(* IEC 61131-3 sources: ST_L/Practice/04_FunctionBlock, 3 files *)

(* ---- 04_01_CounterFB.st ---- *)
(* ============================================================================
 * 文件: 04_01_CounterFB.st
 * 章节: 第7章 - 功能块
 * 描述: 计数器功能块
 * 学习目标: 掌握功能块的定义和实例化
 * ============================================================================ *)

(* ============================================================================
 * 功能块: Counter
 * 功能: 双向计数器，支持递增/递减计数
 * ============================================================================ *)
FUNCTION_BLOCK Counter
VAR_INPUT
    enable : BOOL := TRUE;           // 使能
    preset : INT := 100;             // 预设值
    increment : BOOL;                // 递增触发
    decrement : BOOL;                // 递减触发
    reset : BOOL;                    // 复位
END_VAR

VAR_OUTPUT
    currentValue : INT;              // 当前计数值
    done : BOOL;                     // 计数完成标志
    underflow : BOOL;                // 欠流标志
    overflow : BOOL;                 // 溢出标志
END_VAR

VAR
    lastInc : BOOL := FALSE;         // 上次递增状态
    lastDec : BOOL := FALSE;         // 上次递减状态
    lastReset : BOOL := FALSE;       // 上次复位状态
END_VAR

BEGIN
    (* 检测递增上升沿 *)
    IF increment AND NOT lastInc THEN
        IF enable THEN
            IF currentValue < 32767 THEN
                currentValue := currentValue + 1;
            ELSE
                overflow := TRUE;
            END_IF
        END_IF
    END_IF;

    (* 检测递减上升沿 *)
    IF decrement AND NOT lastDec THEN
        IF enable THEN
            IF currentValue > -32768 THEN
                currentValue := currentValue - 1;
            ELSE
                underflow := TRUE;
            END_IF
        END_IF
    END_IF;

    (* 检测复位上升沿 *)
    IF reset AND NOT lastReset THEN
        currentValue := 0;
        done := FALSE;
        overflow := FALSE;
        underflow := FALSE;
    END_IF;

    (* 更新完成状态 *)
    done := (currentValue >= preset);

    (* 保存上次状态 *)
    lastInc := increment;
    lastDec := decrement;
    lastReset := reset;
END_FUNCTION_BLOCK

(* ============================================================================
 * 功能块: UpCounter (递增计数器简化版)
 * ============================================================================ *)
FUNCTION_BLOCK UpCounter
VAR_INPUT
    enable : BOOL := TRUE;
    preset : INT := 100;
    count : BOOL;                    // 计数脉冲
    reset : BOOL;
END_VAR

VAR_OUTPUT
    q : BOOL;                        // 达到预设值
    cv : INT;                        // 当前值
END_VAR

VAR
    lastCount : BOOL := FALSE;
END_VAR

BEGIN
    (* 边沿检测 *)
    IF count AND NOT lastCount THEN
        IF enable AND NOT q THEN
            cv := cv + 1;
        END_IF
    END_IF;

    (* 复位 *)
    IF reset THEN
        cv := 0;
    END_IF;

    (* 输出 *)
    q := (cv >= preset);
    lastCount := count;
END_FUNCTION_BLOCK

(* ============================================================================
 * 功能块: DownCounter (递减计数器简化版)
 * ============================================================================ *)
FUNCTION_BLOCK DownCounter
VAR_INPUT
    enable : BOOL := TRUE;
    preset : INT := 10;
    count : BOOL;                    // 计数脉冲
    reset : BOOL;
END_VAR

VAR_OUTPUT
    q : BOOL;                        // 计数值减到0
    cv : INT;                        // 当前值
END_VAR

VAR
    lastCount : BOOL := FALSE;
END_VAR

BEGIN
    (* 边沿检测 *)
    IF count AND NOT lastCount THEN
        IF enable AND NOT q THEN
            IF cv > 0 THEN
                cv := cv - 1;
            END_IF
        END_IF
    END_IF;

    (* 复位 *)
    IF reset THEN
        cv := preset;
    END_IF;

    (* 输出 *)
    q := (cv <= 0);
    lastCount := count;
END_FUNCTION_BLOCK

(* ============================================================================
 * 功能块: CounterWithRate (带速率的计数器)
 * ============================================================================ *)
FUNCTION_BLOCK CounterWithRate
VAR_INPUT
    enable : BOOL := TRUE;
    preset : INT := 1000;
    pulse : BOOL;                    // 计数脉冲
    reset : BOOL;
    presetValue : INT;              // 可变预设值
END_VAR

VAR_OUTPUT
    current : INT;                   // 当前值
    done : BOOL;
    rate : REAL;                    // 计数速率 (次/秒)
END_VAR

VAR
    lastPulse : BOOL := FALSE;
    pulseCount : INT := 0;
    lastSecond : TIME := T#0s;
    currentSecond : TIME;
    rateTimer : TON;
END_VAR

BEGIN
    (* 检测脉冲 *)
    IF pulse AND NOT lastPulse THEN
        IF enable THEN
            current := current + 1;
            pulseCount := pulseCount + 1;
        END_IF
    END_IF;

    lastPulse := pulse;

    (* 复位 *)
    IF reset THEN
        current := 0;
        pulseCount := 0;
    END_IF;

    (* 计算速率 *)
    rateTimer(IN := enable, PT := T#1s);
    IF rateTimer.Q THEN
        rate := INT_TO_REAL(pulseCount);
        pulseCount := 0;
        rateTimer(IN := FALSE);
        rateTimer(IN := TRUE, PT := T#1s);
    END_IF;

    (* 完成标志 *)
    IF presetValue > 0 THEN
        done := (current >= presetValue);
    ELSE
        done := (current >= preset);
    END_IF
END_FUNCTION_BLOCK

(* ============================================================================
 * 程序: CounterDemo
 * 功能: 计数器功能块演示
 * ============================================================================ *)
PROGRAM CounterDemo
VAR
    (* 计数器实例 *)
    mainCounter : Counter;
    partCounter : UpCounter;
    batchCounter : DownCounter;
    rateCounter : CounterWithRate;

    (* 输入信号模拟 *)
    bPulse : BOOL := FALSE;
    bButton : BOOL := FALSE;

    (* 输出显示 *)
    iCount : INT;
    bDone : BOOL;
    rRate : REAL;

    (* 测试循环 *)
    i : INT;
END_VAR

BEGIN
    // ==========================================================================
    // 1. 基本计数器演示
    // ==========================================================================

    mainCounter(
        enable := TRUE,
        preset := 10,
        increment := bButton,
        decrement := FALSE,
        reset := FALSE
    );

    // 模拟10次计数
    FOR i := 1 TO 10 DO
        bButton := TRUE;
        mainCounter(
            enable := TRUE,
            preset := 10,
            increment := bButton,
            decrement := FALSE,
            reset := FALSE
        );
        bButton := FALSE;
    END_FOR;

    iCount := mainCounter.currentValue;  // 10
    bDone := mainCounter.done;           // TRUE

    // ==========================================================================
    // 2. 递增计数器演示
    // ==========================================================================

    // 复位
    partCounter(
        enable := TRUE,
        preset := 100,
        count := FALSE,
        reset := TRUE
    );

    // 计数50次
    FOR i := 1 TO 50 DO
        bPulse := TRUE;
        partCounter(
            enable := TRUE,
            preset := 100,
            count := bPulse,
            reset := FALSE
        );
        bPulse := FALSE;
    END_FOR;

    iCount := partCounter.cv;            // 50
    bDone := partCounter.q;             // FALSE

    // ==========================================================================
    // 3. 递减计数器演示
    // ==========================================================================

    batchCounter(
        enable := TRUE,
        preset := 20,
        count := FALSE,
        reset := TRUE
    );

    iCount := batchCounter.cv;          // 20

    // 递减计数
    FOR i := 1 TO 15 DO
        bPulse := TRUE;
        batchCounter(
            enable := TRUE,
            preset := 20,
            count := bPulse,
            reset := FALSE
        );
        bPulse := FALSE;
    END_FOR;

    iCount := batchCounter.cv;          // 5
    bDone := batchCounter.q;            // FALSE

    // 再计5次
    FOR i := 1 TO 5 DO
        bPulse := TRUE;
        batchCounter(
            enable := TRUE,
            preset := 20,
            count := bPulse,
            reset := FALSE
        );
        bPulse := FALSE;
    END_FOR;

    iCount := batchCounter.cv;          // 0
    bDone := batchCounter.q;            // TRUE

    // ==========================================================================
    // 4. 带速率计数器演示
    // ==========================================================================

    rateCounter(
        enable := TRUE,
        preset := 1000,
        pulse := FALSE,
        reset := TRUE,
        presetValue := 0
    );

    rateCounter(
        enable := TRUE,
        preset := 1000,
        pulse := bButton,
        reset := FALSE,
        presetValue := 500
    );

    iCount := rateCounter.current;      // 当前计数
    rRate := rateCounter.rate;          // 速率 (次/秒)

END_PROGRAM

(* ---- 04_02_TimerFB.st ---- *)
(* ============================================================================
 * 文件: 04_02_TimerFB.st
 * 章节: 第7章 - 功能块
 * 描述: 定时器功能块
 * 学习目标: 掌握定时器功能块的编写
 * ============================================================================ *)

(* ============================================================================
 * 功能块: TON - 通电延时定时器
 * 功能: 输入为TRUE时，延时PT后输出Q变为TRUE
 * ============================================================================ *)
FUNCTION_BLOCK TON
VAR_INPUT
    IN : BOOL;    // 触发输入
    PT : TIME;    // 延时时间
END_VAR

VAR_OUTPUT
    Q : BOOL;     // 定时输出
    ET : TIME;    // 已计时时间
END_VAR

VAR
    startTime : TIME;
    running : BOOL := FALSE;
    lastIN : BOOL := FALSE;
END_VAR

BEGIN
    // 检测上升沿
    IF IN AND NOT lastIN THEN
        running := TRUE;
        startTime := TIME();
        Q := FALSE;
    END_IF;

    // 输入变为FALSE，立即复位
    IF NOT IN THEN
        running := FALSE;
        Q := FALSE;
        ET := T#0s;
    END_IF;

    // 计时中
    IF running THEN
        ET := TIME() - startTime;
        IF ET >= PT THEN
            Q := TRUE;
            ET := PT;
        END_IF
    END_IF;

    lastIN := IN;
END_FUNCTION_BLOCK

(* ============================================================================
 * 功能块: TOF - 断电延时定时器
 * 功能: 输入变为FALSE时，延时PT后输出Q变为FALSE
 * ============================================================================ *)
FUNCTION_BLOCK TOF
VAR_INPUT
    IN : BOOL;    // 触发输入
    PT : TIME;    // 延时时间
END_VAR

VAR_OUTPUT
    Q : BOOL;     // 定时输出
    ET : TIME;    // 已计时时间
END_VAR

VAR
    startTime : TIME;
    running : BOOL := FALSE;
    lastIN : BOOL := FALSE;
END_VAR

BEGIN
    // 输入变为TRUE，立即输出TRUE
    IF IN AND NOT lastIN THEN
        Q := TRUE;
        running := FALSE;
        ET := T#0s;
    END_IF;

    // 输入变为FALSE，启动延时
    IF NOT IN AND lastIN THEN
        running := TRUE;
        startTime := TIME();
    END_IF;

    // 计时中
    IF running THEN
        ET := TIME() - startTime;
        IF ET >= PT THEN
            Q := FALSE;
            running := FALSE;
            ET := T#0s;
        END_IF
    END_IF;

    lastIN := IN;
END_FUNCTION_BLOCK

(* ============================================================================
 * 功能块: TP - 脉冲定时器
 * 功能: 每次触发产生固定宽度的脉冲
 * ============================================================================ *)
FUNCTION_BLOCK TP
VAR_INPUT
    IN : BOOL;    // 触发输入
    PT : TIME;    // 脉冲宽度
END_VAR

VAR_OUTPUT
    Q : BOOL;     // 脉冲输出
    ET : TIME;    // 已计时时间
END_VAR

VAR
    startTime : TIME;
    running : BOOL := FALSE;
    lastIN : BOOL := FALSE;
END_VAR

BEGIN
    // 检测上升沿且未运行时启动
    IF IN AND NOT lastIN AND NOT running THEN
        running := TRUE;
        startTime := TIME();
        Q := TRUE;
    END_IF;

    // 计时
    IF running THEN
        ET := TIME() - startTime;
        IF ET >= PT THEN
            Q := FALSE;
            running := FALSE;
            ET := PT;
        END_IF
    ELSE
        ET := T#0s;
    END_IF;

    lastIN := IN;
END_FUNCTION_BLOCK

(* ============================================================================
 * 功能块: TON10ms - 10ms分辨率定时器（软件模拟）
 * 功能: 适用于不支持TIME类型的系统
 * ============================================================================ *)
FUNCTION_BLOCK TON10ms
VAR_INPUT
    IN : BOOL;
    PTms : INT;    // 延时时间（毫秒）
END_VAR

VAR_OUTPUT
    Q : BOOL;
    ETms : INT;    // 已计时时间（毫秒）
END_VAR

VAR
    startTick : INT;
    running : BOOL := FALSE;
    lastIN : BOOL := FALSE;
    currentTick : INT;
END_VAR

BEGIN
    // 检测上升沿
    IF IN AND NOT lastIN THEN
        running := TRUE;
        startTick := currentTick;
        Q := FALSE;
    END_IF;

    // 输入变为FALSE，立即复位
    IF NOT IN THEN
        running := FALSE;
        Q := FALSE;
        ETms := 0;
    END_IF;

    // 计时中
    IF running THEN
        ETms := (currentTick - startTick) * 10;  // 假设每个tick为10ms
        IF ETms >= PTms THEN
            Q := TRUE;
            ETms := PTms;
        END_IF
    END_IF;

    lastIN := IN;
END_FUNCTION_BLOCK

(* ============================================================================
 * 功能块: Blinker - 闪烁定时器
 * 功能: 产生连续闪烁信号
 * ============================================================================ *)
FUNCTION_BLOCK Blinker
VAR_INPUT
    enable : BOOL;
    period : TIME := T#1s;    // 闪烁周期
END_VAR

VAR_OUTPUT
    Q : BOOL;                 // 闪烁输出
END_VAR

VAR
    timer : TON;
    toggle : BOOL := FALSE;
END_VAR

BEGIN
    IF enable THEN
        timer(IN := NOT timer.Q, PT := period);
        IF timer.Q THEN
            toggle := NOT toggle;
        END_IF;
        Q := toggle;
    ELSE
        Q := FALSE;
        toggle := FALSE;
        timer(IN := FALSE);
    END_IF
END_FUNCTION_BLOCK

(* ============================================================================
 * 功能块: Watchdog - 看门狗定时器
 * 功能: 监控信号是否正常
 * ============================================================================ *)
FUNCTION_BLOCK Watchdog
VAR_INPUT
    IN : BOOL;                // 被监控信号
    timeout : TIME := T#5s;   // 超时时间
    reset : BOOL;             // 手动复位
END_VAR

VAR_OUTPUT
    Q : BOOL;                 // 超时标志
    ET : TIME;                // 已超时时间
END_VAR

VAR
    timer : TON;
END_VAR

BEGIN
    // 监控信号
    timer(IN := NOT IN, PT := timeout);
    Q := timer.Q;
    ET := timer.ET;

    // 手动复位
    IF reset THEN
        timer(IN := FALSE);
        Q := FALSE;
    END_IF
END_FUNCTION_BLOCK

(* ============================================================================
 * 程序: TimerDemo
 * 功能: 定时器功能块演示
 * ============================================================================ *)
PROGRAM TimerDemo
VAR
    (* 定时器实例 *)
    startDelay : TON;          // 启动延时
    stopDelay : TOF;           // 停止延时
    pulseTimer : TP;           // 脉冲定时器
    warningBlink : Blinker;    // 警告闪烁
    motorWatchdog : Watchdog;   // 电机看门狗

    (* 输入信号 *)
    bStartButton : BOOL := TRUE;
    bStopButton : BOOL := FALSE;
    bMotorRunning : BOOL := FALSE;
    bFaultPresent : BOOL := FALSE;

    (* 输出 *)
    bMotor : BOOL;
    bWarningLight : BOOL;
    bWatchdogFault : BOOL;

    (* 状态显示 *)
    tElapsed : TIME;
END_VAR

BEGIN
    // ==========================================================================
    // 1. 启动延时 (TON)
    // ==========================================================================
    // 按下启动按钮后，延时2秒启动电机

    startDelay(
        IN := bStartButton,
        PT := T#2s
    );

    bMotor := startDelay.Q;
    tElapsed := startDelay.ET;

    // ==========================================================================
    // 2. 停止延时 (TOF)
    // ==========================================================================
    // 松开停止按钮后，延时3秒停止电机（用于平滑停止）

    stopDelay(
        IN := bStopButton,
        PT := T#3s
    );

    // 注意: TOF的逻辑是输入FALSE时延时
    // 这里需要反向逻辑

    // ==========================================================================
    // 3. 脉冲定时器 (TP)
    // ==========================================================================
    // 产生一个500ms的脉冲

    pulseTimer(
        IN := bStartButton,
        PT := T#500ms
    );

    // pulseTimer.Q 会在按下按钮时产生500ms脉冲

    // ==========================================================================
    // 4. 闪烁定时器
    // ==========================================================================
    // 故障时警告灯以1Hz闪烁

    warningBlink(
        enable := bFaultPresent,
        period := T#1s
    );

    bWarningLight := warningBlink.Q;

    // ==========================================================================
    // 5. 看门狗定时器
    // ==========================================================================
    // 监控电机运行信号，5秒无信号则报警

    motorWatchdog(
        IN := bMotorRunning,
        timeout := T#5s,
        reset := FALSE
    );

    bWatchdogFault := motorWatchdog.Q;

    // ==========================================================================
    // 综合应用示例
    // ==========================================================================

    // 使用TON实现延时启动
    startDelay(IN := bStartButton, PT := T#1s);

    // 组合使用: 启动延时 + 脉冲指示
    IF startDelay.Q AND NOT bMotor THEN
        pulseTimer(IN := TRUE, PT := T#200ms);
        bMotor := TRUE;
    END_IF

    // 故障时闪烁
    IF bFaultPresent THEN
        warningBlink(enable := TRUE, period := T#500ms);
        bWarningLight := warningBlink.Q;
    ELSE
        warningBlink(enable := FALSE);
        bWarningLight := FALSE;
    END_IF

END_PROGRAM

(* ---- 04_03_EdgeDetect.st ---- *)
(* ============================================================================
 * 文件: 04_03_EdgeDetect.st
 * 章节: 第7章 - 功能块
 * 描述: 边沿检测功能块
 * 学习目标: 掌握边沿检测的原理和实现
 * ============================================================================ *)

(* ============================================================================
 * 功能块: R_TRIG - 上升沿检测
 * 功能: 检测信号从FALSE变为TRUE的时刻
 * ============================================================================ *)
FUNCTION_BLOCK R_TRIG
VAR_INPUT
    CLK : BOOL;    // 输入信号
END_VAR

VAR_OUTPUT
    Q : BOOL;      // 上升沿脉冲输出
END_VAR

VAR
    lastCLK : BOOL := FALSE;
END_VAR

BEGIN
    // 上升沿条件: 当前=TRUE 且 上次=FALSE
    Q := CLK AND NOT lastCLK;
    lastCLK := CLK;
END_FUNCTION_BLOCK

(* ============================================================================
 * 功能块: F_TRIG - 下降沿检测
 * 功能: 检测信号从TRUE变为FALSE的时刻
 * ============================================================================ *)
FUNCTION_BLOCK F_TRIG
VAR_INPUT
    CLK : BOOL;    // 输入信号
END_VAR

VAR_OUTPUT
    Q : BOOL;      // 下降沿脉冲输出
END_VAR

VAR
    lastCLK : BOOL := FALSE;
END_VAR

BEGIN
    // 下降沿条件: 当前=FALSE 且 上次=TRUE
    Q := NOT CLK AND lastCLK;
    lastCLK := CLK;
END_FUNCTION_BLOCK

(* ============================================================================
 * 功能块: CounterFB - 基于边沿的计数器
 * 功能: 使用边沿检测实现脉冲计数
 * ============================================================================ *)
FUNCTION_BLOCK CounterFB
VAR_INPUT
    clock : BOOL;              // 时钟输入
    reset : BOOL;              // 复位输入
    preset : INT := 100;       // 预设值
    direction : BOOL := TRUE;   // 方向: TRUE=递增, FALSE=递减
END_VAR

VAR_OUTPUT
    Q : BOOL;                   // 达到预设
    underflow : BOOL;           // 欠流
    cv : INT;                   // 当前值
END_VAR

VAR
    risingEdge : R_TRIG;
    lastReset : BOOL := FALSE;
END_VAR

BEGIN
    // 检测复位上升沿
    IF reset AND NOT lastReset THEN
        cv := 0;
    END_IF;
    lastReset := reset;

    // 检测时钟上升沿
    risingEdge(CLK := clock);
    IF risingEdge.Q THEN
        IF direction THEN
            // 递增计数
            IF cv < 32767 THEN
                cv := cv + 1;
            END_IF;
        ELSE
            // 递减计数
            IF cv > -32768 THEN
                cv := cv - 1;
            END_IF;
        END_IF
    END_IF;

    // 输出状态
    Q := (cv >= preset);
    underflow := (cv <= 0);

END_FUNCTION_BLOCK

(* ============================================================================
 * 功能块: OneShot - 单次触发
 * 功能: 信号第一次变为TRUE时输出TRUE，之后保持FALSE直到复位
 * ============================================================================ *)
FUNCTION_BLOCK OneShot
VAR_INPUT
    trigger : BOOL;    // 触发信号
    reset : BOOL;     // 复位信号
END_VAR

VAR_OUTPUT
    Q : BOOL;         // 单次输出
END_VAR

VAR
    armed : BOOL := TRUE;  //  armed = TRUE 时可以触发
    lastTrigger : BOOL := FALSE;
END_VAR

BEGIN
    // 检测触发上升沿
    IF trigger AND NOT lastTrigger THEN
        IF armed THEN
            Q := TRUE;
            armed := FALSE;
        END_IF
    END_IF;

    // 复位
    IF reset THEN
        Q := FALSE;
        armed := TRUE;
    END_IF;

    lastTrigger := trigger;
END_FUNCTION_BLOCK

(* ============================================================================
 * 功能块: Toggle - 翻转触发
 * 功能: 每次触发时翻转输出状态
 * ============================================================================ *)
FUNCTION_BLOCK Toggle
VAR_INPUT
    trigger : BOOL;    // 触发信号
    reset : BOOL;      // 复位信号
END_VAR

VAR_OUTPUT
    Q : BOOL;          // 翻转输出
END_VAR

VAR
    lastTrigger : BOOL := FALSE;
END_VAR

BEGIN
    // 检测触发上升沿
    IF trigger AND NOT lastTrigger THEN
        Q := NOT Q;
    END_IF;

    // 复位
    IF reset THEN
        Q := FALSE;
    END_IF;

    lastTrigger := trigger;
END_FUNCTION_BLOCK

(* ============================================================================
 * 功能块: PulseGenerator - 脉冲生成器
 * 功能: 产生指定数量的脉冲
 * ============================================================================ *)
FUNCTION_BLOCK PulseGenerator
VAR_INPUT
    trigger : BOOL;        // 触发信号
    pulseCount : INT := 5; // 脉冲数量
    pulseWidth : TIME := T#100ms;  // 脉冲宽度
END_VAR

VAR_OUTPUT
    Q : BOOL;              // 脉冲输出
    busy : BOOL;           // 工作中
    done : BOOL;           // 完成
END_VAR

VAR
    edgeDetect : R_TRIG;
    timer : TP;
    remaining : INT := 0;
    lastTrigger : BOOL := FALSE;
    generating : BOOL := FALSE;
END_VAR

BEGIN
    // 检测触发
    edgeDetect(CLK := trigger);
    IF edgeDetect.Q AND NOT generating THEN
        remaining := pulseCount;
        generating := TRUE;
        done := FALSE;
    END_IF;

    // 生成脉冲
    IF generating THEN
        busy := TRUE;

        // 生成脉冲
        timer(IN := (remaining > 0), PT := pulseWidth);
        Q := timer.Q;

        // 计数
        IF timer.Q AND (remaining > 0) THEN
            remaining := remaining - 1;
        END_IF;

        // 完成
        IF remaining <= 0 THEN
            generating := FALSE;
            busy := FALSE;
            done := TRUE;
            Q := FALSE;
        END_IF
    ELSE
        busy := FALSE;
        done := FALSE;
        Q := FALSE;
        timer(IN := FALSE);
    END_IF;

    lastTrigger := trigger;
END_FUNCTION_BLOCK

(* ============================================================================
 * 功能块: Debounce - 防抖模块
 * 功能: 对输入信号进行防抖处理
 * ============================================================================ *)
FUNCTION_BLOCK Debounce
VAR_INPUT
    signal : BOOL;                 // 输入信号
    debounceTime : TIME := T#50ms; // 防抖时间
END_VAR

VAR_OUTPUT
    Q : BOOL;                      // 去抖后输出
END_VAR

VAR
    timer : TON;
    lastSignal : BOOL := FALSE;
END_VAR

BEGIN
    // 状态改变时启动定时器
    IF signal <> lastSignal THEN
        timer(IN := TRUE, PT := debounceTime);
    END_IF;

    // 定时结束且信号稳定
    IF timer.Q THEN
        Q := signal;
    END_IF;

    // 定时结束前保持原状态
    IF NOT timer.Q AND timer.ET > T#0ms THEN
        // 等待中，保持原状态
    END_IF;

    // 信号稳定后复位定时器
    IF signal = lastSignal THEN
        timer(IN := FALSE);
    END_IF;

    lastSignal := signal;
END_FUNCTION_BLOCK

(* ============================================================================
 * 程序: EdgeDetectionDemo
 * 功能: 边沿检测功能块演示
 * ============================================================================ *)
PROGRAM EdgeDetectionDemo
VAR
    (* 边沿检测实例 *)
    sensorRising : R_TRIG;
    buttonRising : R_TRIG;
    sensorFalling : F_TRIG;

    (* 计数器实例 *)
    partCounter : CounterFB;
    cycleCounter : CounterFB;

    (* 其他功能块实例 *)
    motorToggle : Toggle;
    startOneShot : OneShot;
    pulseGen : PulseGenerator;
    inputDebounce : Debounce;

    (* 输入信号 *)
    bSensor : BOOL := FALSE;
    bButton : BOOL := FALSE;
    bReset : BOOL := FALSE;

    (* 输出 *)
    iPartCount : INT;
    bMotorRunning : BOOL;
    iPulseOutput : BOOL;
    bDebounced : BOOL;

    (* 边沿信号 *)
    bSensorEdge : BOOL;
    bButtonEdge : BOOL;

    (* 循环计数 *)
    i : INT;
END_VAR

BEGIN
    // ==========================================================================
    // 1. 上升沿检测
    // ==========================================================================

    sensorRising(CLK := bSensor);
    bSensorEdge := sensorRising.Q;

    // 检测到上升沿时计数
    IF bSensorEdge THEN
        iPartCount := iPartCount + 1;
    END_IF

    // ==========================================================================
    // 2. 下降沿检测
    // ==========================================================================

    sensorFalling(CLK := bSensor);
    // bSensorEdge := sensorFalling.Q; // 下降沿检测

    // ==========================================================================
    // 3. 翻转触发
    // ==========================================================================

    motorToggle(trigger := bButton, reset := bReset);
    bMotorRunning := motorToggle.Q;

    // ==========================================================================
    // 4. 单次触发
    // ==========================================================================

    startOneShot(trigger := bButton, reset := bReset);
    // startOneShot.Q 只在第一次触发时为TRUE

    // ==========================================================================
    // 5. 防抖
    // ==========================================================================

    inputDebounce(
        signal := bSensor,
        debounceTime := T#50ms
    );
    bDebounced := inputDebounce.Q;

    // ==========================================================================
    // 6. 脉冲生成器
    // ==========================================================================

    pulseGen(
        trigger := bButton,
        pulseCount := 5,
        pulseWidth := T#100ms
    );
    iPulseOutput := pulseGen.Q;

    // ==========================================================================
    // 7. 组合应用示例
    // ==========================================================================

    // 检测启动按钮上升沿，计数
    buttonRising(CLK := bButton);
    IF buttonRising.Q THEN
        partCounter(
            clock := TRUE,
            reset := bReset,
            preset := 100,
            direction := TRUE
        );
    END_IF

    iPartCount := partCounter.cv;

END_PROGRAM
